# EPICS substitutions: LINMOT/LINMOT-IOC-01App/Db/motorSim.substitutions
#file $(MOTOR)/db/motor.db {
#
#pattern {P,    M,         DTYP,      DESC,   EGU,  DIR,  VELO,  VBAS, ACCL, BDST, BVEL, BACC,    MRES,    ERES, UEIP, PREC, DHLM, DLLM, INIT, C, S, MOTORSIM }
#{"\$(P)", "\$(M)", "Motor Simulation", "\$(NAME) (LINMOT)",    "degree",  "Pos",  "\$(VELO)",   1,  "\$(ACCL)",    0,    1,   0,   "\$(MRES)",   "\$(ERES)", "\$(UEIP)",    3,   "\$(DHLM)",   "\$(DLLM)",  "", "\$(C)", "\$(S)", "motorSim" }
#
#}

file $(MOTOR)/db/asyn_motor.db {

pattern {P,    M,         DTYP,      DESC,   EGU,  DIR,  VELO,  VBAS, ACCL, BDST, BVEL, BACC,    MRES,    ERES, UEIP, PREC, DHLM, DLLM, INIT, C, S, MOTORSIM, PORT, ADDR }
{"\$(P)", "\$(M)", "asynMotor", "\$(NAME) (LINMOT)",    "\$(EGU)",  "Pos",  "\$(VELO)",   1,  "\$(ACCL)",    0,    1,   0,   "\$(MRES)",   "\$(ERES)", "\$(UEIP)",    3,   "\$(DHLM)",   "\$(DLLM)",  "", "\$(C)", "\$(S)", "motorSim", "motorSim", "0" }

}
